(* Logix 5000 project; controller V34L73S_S00 1756-L85E rev 34.11; software revision 34.00 *)

TASK MainTask (continuous, watchdog 500 ms) : MainProgram
TASK SafetyTask (periodic, rate 20 ms, priority 10, watchdog 20 ms) : SafetyProgram

MODULES
   Local : 1756-L85E (ICP 13, rev 34.11)
END_MODULES

TYPE UserDefinedType :
STRUCT
   BOOL : BOOL;
   DINT : DINT;
   TIMER : TIMER;
   STRING : STRING;
   StringArray : STRING[2];
END_STRUCT
END_TYPE

VAR_GLOBAL   (* controller tags *)
   Controller_Alias_Bool : ALIAS FOR Controller_UDTArray[0,0,1].BOOL;
   Controller_alias_dint : ALIAS FOR Controller_UDTArray[1,0,0].DINT;
   Controller_Alias_String : ALIAS FOR Controller_STRINGARRAY[1,0];
   Controller_Alias_Timer : ALIAS FOR Controller_Timer_Array[2,2,2];
   Controller_BOOL : BOOL;
   Controller_Bool_Array : BOOL[32];
   Controller_DINT : DINT := 17;
   Controller_LINT : LINT := 48;
   Controller_REAL : REAL := 27.678343;
   Controller_Safety_DINT : DINT := 2;
   Controller_SINT : SINT := 62;
   Controller_STRING : STRING := 'yo';
   Controller_STRINGARRAY : STRING[2,2] := ([0,0] := 'hi', [1,0] := 'zzzzzz', [1,1] := 'test3');
   Controller_TIMER : TIMER := (PRE := 1500, ACC := 1500, EN := 1, DN := 1);
   Controller_Timer_Array : TIMER[4,4,4] := ([2,2,2].PRE := 4000, [2,2,2].ACC := 4000, [2,2,2].EN := 1, [2,2,2].DN := 1);
   Controller_UDT : UserDefinedType := (DINT := 37, TIMER.PRE := 8000, TIMER.ACC := 1387, TIMER.EN := 1, TIMER.TT := 1, STRING := 'no', StringArray[0] := 'yes1', StringArray[1] := 'test4');
   Controller_UDTArray : UserDefinedType[2,2,2] := ([0,0,0].DINT := -1, [0,0,0].TIMER.PRE := 9000, [0,0,0].TIMER.ACC := 8330, [0,0,0].TIMER.EN := 1, [0,0,0].TIMER.TT := 1, [0,0,0].STRING := 'test', [0,0,0].StringArray[0] := 'test21', [0,0,0].StringArray[1] := 'test5', [1,0,0].DINT := -1, [1,0,1].TIMER.PRE := 6000, [1,0,1].TIMER.ACC := 3346, [1,0,1].TIMER.EN := 1, [1,0,1].TIMER.TT := 1, [1,0,1].STRING := 'test', [1,0,1].StringArray[0] := 'test23', [1,0,1].StringArray[1] := 'test3');
END_VAR

PROGRAM MainProgram   (* main routine MainRoutine *)
VAR
   MainProgram_Alias_Bool : ALIAS FOR MainProgram_UDTArray[0,0,1].BOOL;
   MainProgram_Alias_Bools_DINT : ALIAS FOR MainProgram_DINT;
   MainProgram_alias_dint : ALIAS FOR MainProgram_UDTArray[1,0,0].DINT;
   MainProgram_Alias_String : ALIAS FOR MainProgram_STRINGARRAY[1,0];
   MainProgram_Alias_Timer : ALIAS FOR MainProgram_Timer_Array[2,2,2];
   MainProgram_BOOL : BOOL;
   MainProgram_Bool_Array : BOOL[32];
   MainProgram_DINT : DINT := 30;
   MainProgram_LINT : LINT := 4;
   MainProgram_REAL : REAL := 1.45874;
   MainProgram_Safety_DINT : DINT;
   MainProgram_SINT : SINT := -9;
   MainProgram_STRING : STRING;
   MainProgram_STRINGARRAY : STRING[2,2];
   MainProgram_TIMER : TIMER := (PRE := 2000, ACC := 2000, EN := 1, DN := 1);
   MainProgram_Timer_Array : TIMER[4,4,4] := ([2,2,2].PRE := 4000, [2,2,2].ACC := 4000, [2,2,2].EN := 1, [2,2,2].DN := 1);
   MainProgram_UDT : UserDefinedType := (TIMER.PRE := 8000, TIMER.ACC := 1444, TIMER.EN := 1, TIMER.TT := 1);
   MainProgram_UDTArray : UserDefinedType[2,2,2] := ([0,0,0].TIMER.PRE := 6000, [0,0,0].TIMER.ACC := 5397, [0,0,0].TIMER.EN := 1, [0,0,0].TIMER.TT := 1, [1,0,1].TIMER.PRE := 6000, [1,0,1].TIMER.ACC := 3413, [1,0,1].TIMER.EN := 1, [1,0,1].TIMER.TT := 1);
END_VAR

ROUTINE MainRoutine   (* ladder *)
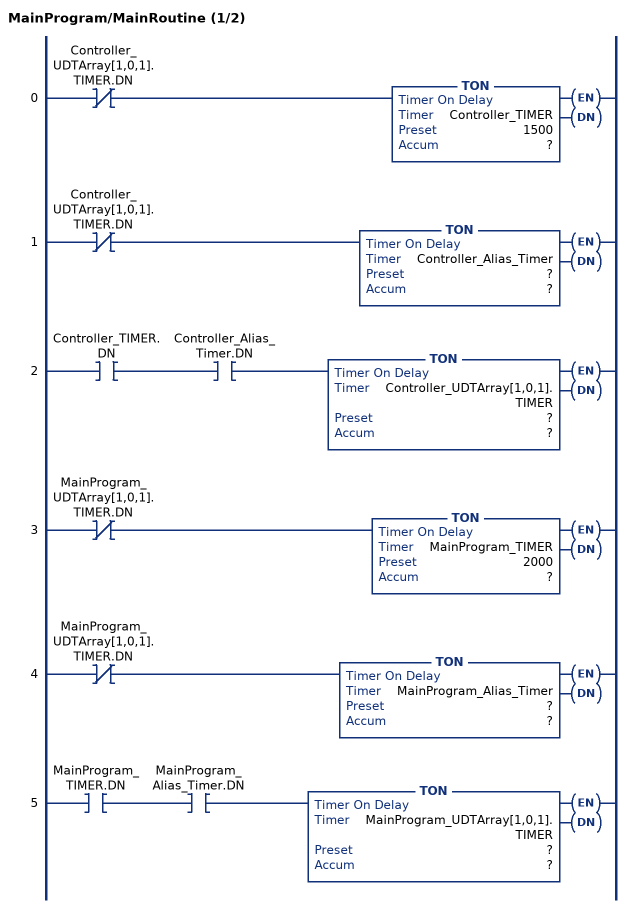
   0: XIO(Controller_UDTArray[1,0,1].TIMER.DN)TON(Controller_TIMER,?,?);
   1: XIO(Controller_UDTArray[1,0,1].TIMER.DN)TON(Controller_Alias_Timer,?,?);
   2: XIC(Controller_TIMER.DN)XIC(Controller_Alias_Timer.DN)TON(Controller_UDTArray[1,0,1].TIMER,?,?);
   3: XIO(MainProgram_UDTArray[1,0,1].TIMER.DN)TON(MainProgram_TIMER,?,?);
   4: XIO(MainProgram_UDTArray[1,0,1].TIMER.DN)TON(MainProgram_Alias_Timer,?,?);
   5: XIC(MainProgram_TIMER.DN)XIC(MainProgram_Alias_Timer.DN)TON(MainProgram_UDTArray[1,0,1].TIMER,?,?);
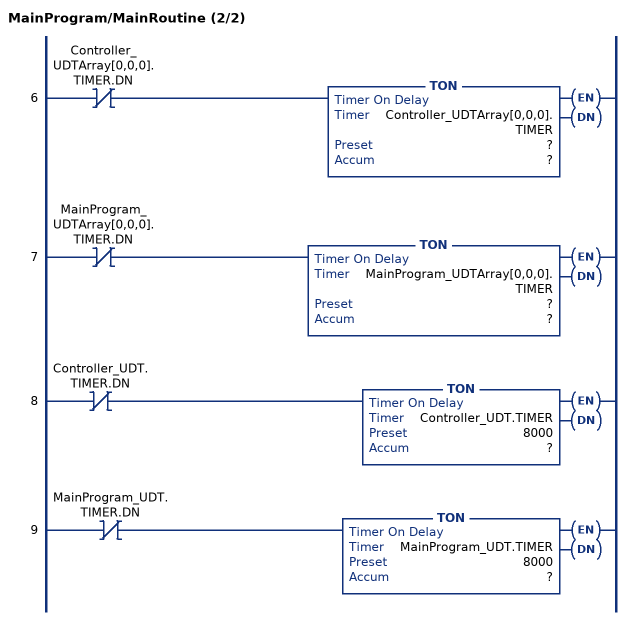
   6: XIO(Controller_UDTArray[0,0,0].TIMER.DN)TON(Controller_UDTArray[0,0,0].TIMER,?,?);
   7: XIO(MainProgram_UDTArray[0,0,0].TIMER.DN)TON(MainProgram_UDTArray[0,0,0].TIMER,?,?);
   8: XIO(Controller_UDT.TIMER.DN)TON(Controller_UDT.TIMER,?,?);
   9: XIO(MainProgram_UDT.TIMER.DN)TON(MainProgram_UDT.TIMER,?,?);
END_ROUTINE
END_PROGRAM

PROGRAM SafetyProgram   (* main routine MainRoutine *)
VAR
   SafetyProgram_Alias_Bool : ALIAS FOR SafetyProgram_UDTArray[0,0,1].BOOL;
   SafetyProgram_Alias_Bools_DINT : ALIAS FOR SafetyProgram_DINT;
   SafetyProgram_alias_dint : ALIAS FOR SafetyProgram_UDTArray[1,0,0].DINT;
   SafetyProgram_Alias_String : ALIAS FOR SafetyProgram_STRINGARRAY[1,0];
   SafetyProgram_Alias_Timer : ALIAS FOR SafetyProgram_Timer_Array[2,2,2];
   SafetyProgram_BOOL : BOOL;
   SafetyProgram_Bool_Array : BOOL[32];
   SafetyProgram_DINT : DINT;
   SafetyProgram_REAL : REAL;
   SafetyProgram_Safety_DINT : DINT;
   SafetyProgram_SINT : SINT;
   SafetyProgram_STRING : STRING;
   SafetyProgram_STRINGARRAY : STRING[2,2];
   SafetyProgram_TIMER : TIMER := (PRE := 9000, ACC := 2840, EN := 1, TT := 1);
   SafetyProgram_Timer_Array : TIMER[4,4,4] := ([2,2,2].PRE := 4000, [2,2,2].ACC := 2840, [2,2,2].EN := 1, [2,2,2].TT := 1);
   SafetyProgram_UDT : UserDefinedType := (TIMER.PRE := 8000, TIMER.ACC := 800, TIMER.EN := 1, TIMER.TT := 1);
   SafetyProgram_UDTArray : UserDefinedType[2,2,2] := ([0,0,0].TIMER.PRE := 9000, [0,0,0].TIMER.ACC := 7120, [0,0,0].TIMER.EN := 1, [0,0,0].TIMER.TT := 1, [1,0,1].TIMER.PRE := 6000);
END_VAR

ROUTINE MainRoutine   (* ladder *)
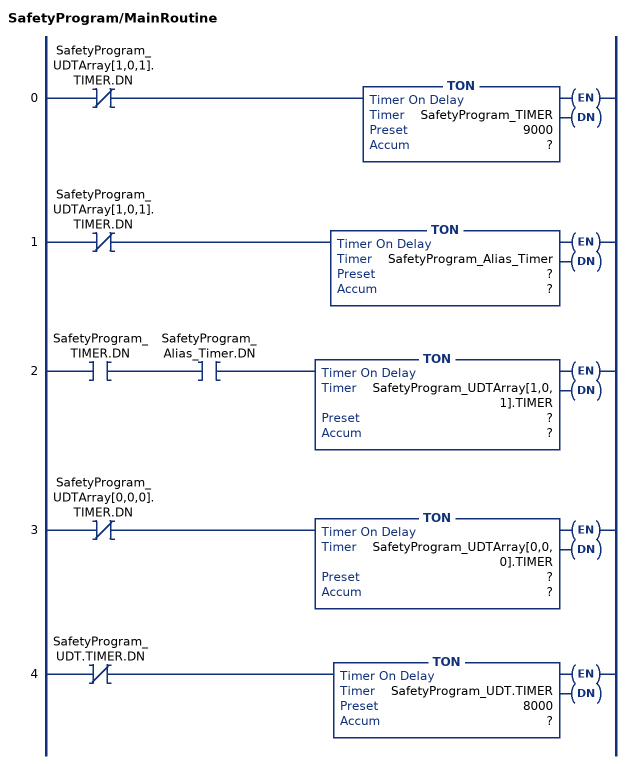
   0: XIO(SafetyProgram_UDTArray[1,0,1].TIMER.DN)TON(SafetyProgram_TIMER,?,?);
   1: XIO(SafetyProgram_UDTArray[1,0,1].TIMER.DN)TON(SafetyProgram_Alias_Timer,?,?);
   2: XIC(SafetyProgram_TIMER.DN)XIC(SafetyProgram_Alias_Timer.DN)TON(SafetyProgram_UDTArray[1,0,1].TIMER,?,?);
   3: XIO(SafetyProgram_UDTArray[0,0,0].TIMER.DN)TON(SafetyProgram_UDTArray[0,0,0].TIMER,?,?);
   4: XIO(SafetyProgram_UDT.TIMER.DN)TON(SafetyProgram_UDT.TIMER,?,?);
END_ROUTINE
END_PROGRAM
